// TIA Portal V18 export
VAR_GLOBAL   // PLC tag table "默认变量表"
   Room1_ES1 AT %I200.0 : Bool;
   Room1_ES2 AT %I200.1 : Bool;
   Room1_ES3 AT %I200.2 : Bool;
   Room1_ES4 AT %I200.3 : Bool;
   Room1_ES5 AT %I206.0 : Bool;
   Room1Control_ES6 AT %I206.1 : Bool;
   "Room1_Key1.1" AT %I206.2 : Bool;
   "Room1Control_Key1.1" AT %I206.3 : Bool;
   "Room1_door1.1" AT %I212.0 : Bool;
   Room2_ES1 AT %I218.0 : Bool;
   Room2_ES2 AT %I218.1 : Bool;
   Room2_ES3 AT %I218.2 : Bool;
   Room2_ES4 AT %I218.3 : Bool;
   Room2_ES5 AT %I224.0 : Bool;
   Room2Control_ES6 AT %I224.1 : Bool;
   "Room2_Key1.1" AT %I224.2 : Bool;
   "Room2Control_Key1.1" AT %I224.3 : Bool;
   "Room2_door1.1" AT %I230.0 : Bool;
   ACC_ES1 AT %I236.0 : Bool;
   ACC_ES2 AT %I236.1 : Bool;
   ACC_ES3 AT %I236.2 : Bool;
   ACC_ES4 AT %I236.3 : Bool;
   "ACC_Key1.1" AT %I242.2 : Bool;
   "ACCControl_Key1.1" AT %I242.3 : Bool;
   "ACC_door1.1" AT %I248.0 : Bool;
   "ACC_door2.1" AT %I248.1 : Bool;
   VerticalBeam_ES1 AT %I254.0 : Bool;   // vertical beam ES
   VerticalBeam_ES2 AT %I254.1 : Bool;
   VerticalBeam_ES3 AT %I254.2 : Bool;
   VerticalBeam_ES4 AT %I254.3 : Bool;
   "VerticalBeam_Key1.1" AT %I260.2 : Bool;
   "VerticalBeamControl_Key1.1" AT %I260.3 : Bool;
   "VerticalBeam_door1.1" AT %I266.0 : Bool;
   "VerticalBeam_door2.1" AT %I266.1 : Bool;
   Room1_SB1 AT %I100.0 : Bool;   // 搜索清场按钮1
   Room1_SB2 AT %I100.1 : Bool;
   Room2_SB1 AT %I100.4 : Bool;
   Room2_SB2 AT %I100.5 : Bool;
   ACC_SB1 AT %I101.0 : Bool;
   ACC_SB2 AT %I101.1 : Bool;
   VerticalBeam_SB1 AT %I101.4 : Bool;
   VerticalBeam_SB2 AT %I101.5 : Bool;
   ACC_Ready AT %I102.0 : Bool;
   ACC_Run AT %I102.1 : Bool;
   ACC_StopBeam AT %I102.2 : Bool;
   ACC_Stop AT %I102.3 : Bool;
   ACC_Fault AT %I102.4 : Bool;
   ACC_Mode1 AT %I102.5 : Bool;   // 治疗室1、加速器2、垂直束
   ACC_Mode2 AT %I102.6 : Bool;   // 治疗室2、加速器2、垂直束
   ACC_Mode3 AT %I102.7 : Bool;   // 加速器2、垂直束
   EnvironmentalMonitoring1 AT %I103.4 : Bool;
   EnvironmentalMonitoring2 AT %I103.5 : Bool;
   EnvironmentalMonitoring3 AT %I103.6 : Bool;
   EnvironmentalMonitoring4 AT %I103.7 : Bool;
   Room1_AudibleAlarm AT %Q100.0 : Bool;
   Room1_StrobeLamp1 AT %Q100.1 : Bool;
   Room1_StrobeLamp2 AT %Q100.2 : Bool;
   Room1_Red AT %Q100.5 : Bool;   // 禁止进入指示灯
   Room1_Yellow AT %Q100.6 : Bool;   // 限制进入指示灯
   Room1_Green AT %Q100.7 : Bool;   // 控制进入指示灯
   Room1_Door1NoEntry AT %Q101.0 : Bool;   // 门禁1禁止进入
   Room1_Door1RestrictedEntry AT %Q101.1 : Bool;   // 门禁1限制进入
   Room1_Door1ControlEntry AT %Q101.2 : Bool;   // 门禁1控制进入
   "Room1_door1.2" AT %I212.4 : Bool;
   "Room1_Key1.2" AT %I206.6 : Bool;
   "Room1Control_Key1.2" AT %I206.7 : Bool;
   "Room2_Key1.2" AT %I224.6 : Bool;
   "Room2Control_Key1.2" AT %I224.7 : Bool;
   "Room2_door1.2" AT %I230.4 : Bool;
   "ACC_Key1.2" AT %I242.6 : Bool;
   "ACCControl_Key1.2" AT %I242.7 : Bool;
   "VerticalBeam_Key1.2" AT %I260.6 : Bool;
   "VerticalBeamControl_Key1.2" AT %I260.7 : Bool;
   "VerticalBeam_door1.2" AT %I266.4 : Bool;
   "VerticalBeam_door2.2" AT %I266.5 : Bool;
   "ACC_door1.2" AT %I248.4 : Bool;
   "ACC_door2.2" AT %I248.5 : Bool;
   ACC_Interlock1 AT %Q400.0 : Bool;
   ACC_Interlock2 AT %Q400.1 : Bool;
   RF_Interlock1 AT %Q400.2 : Bool;
   RF_Interlock2 AT %Q400.3 : Bool;
   IonSource_Interlock1 AT %Q400.4 : Bool;
   IonSource_Interlock2 AT %Q400.5 : Bool;
   MIS__Interlock1 AT %Q400.6 : Bool;
   MIS__Interlock2 AT %Q400.7 : Bool;
   Room1_ES1_ValueStatus AT %I201.0 : Bool;
   Room1_ES2_ValueStatus AT %I201.1 : Bool;
   Room1_ES3_ValueStatus AT %I201.2 : Bool;
   Room1_ES4_ValueStatus AT %I201.3 : Bool;
   Room1_ES5_ValueStatus AT %I207.0 : Bool;
   Room1Control_ES6_ValueStatus AT %I207.1 : Bool;
   "Room1_Key1.1_ValueStatus" AT %I207.2 : Bool;
   "Room1Control_Key1.1_ValueStatus" AT %I207.3 : Bool;
   "Room1_Key1.2_ValueStatus" AT %I207.6 : Bool;
   "Room1Control_Key1.2_ValueStatus" AT %I207.7 : Bool;
   "Room1_door1.1_ValueStatus" AT %I213.0 : Bool;
   "Room1_door1.2_ValueStatus" AT %I213.4 : Bool;
   Room2_ES1_ValueStatus AT %I219.0 : Bool;
   Room2_ES2_ValueStatus AT %I219.1 : Bool;
   Room2_ES3_ValueStatus AT %I219.2 : Bool;
   Room2_ES4_ValueStatus AT %I219.3 : Bool;
   Room2_ES5_ValueStatus AT %I225.0 : Bool;
   Room2Control_ES6_ValueStatus AT %I225.1 : Bool;
   "Room2_Key1.1_ValueStatus" AT %I225.2 : Bool;
   "Room2Control_Key1.1_ValueStatus" AT %I225.3 : Bool;
   "Room2_Key1.2_ValueStatus" AT %I225.6 : Bool;
   "Room2Control_Key1.2_ValueStatus" AT %I225.7 : Bool;
   "Room2_door1.1_ValueStatus" AT %I231.0 : Bool;
   "Room2_door1.2_ValueStatus" AT %I231.4 : Bool;
   ACC_ES1_ValueStatus AT %I237.0 : Bool;
   ACC_ES2_ValueStatus AT %I237.1 : Bool;
   ACC_ES3_ValueStatus AT %I237.2 : Bool;
   ACC_ES4_ValueStatus AT %I237.3 : Bool;
   "ACC_Key1.1_ValueStatus" AT %I243.2 : Bool;
   "ACCControl_Key1.1_ValueStatus" AT %I243.3 : Bool;
   "ACC_Key1.2_ValueStatus" AT %I243.6 : Bool;
   "ACCControl_Key1.2_ValueStatus" AT %I243.7 : Bool;
   "ACC_door1.1_ValueStatus" AT %I249.0 : Bool;
   "ACC_door2.1_ValueStatus" AT %I249.1 : Bool;
   "ACC_door1.2_ValueStatus" AT %I249.4 : Bool;
   "ACC_door2.2_ValueStatus" AT %I249.5 : Bool;
   VerticalBeam_ES1_ValueStatus AT %I255.0 : Bool;
   VerticalBeam_ES2_ValueStatus AT %I255.1 : Bool;
   VerticalBeam_ES3_ValueStatus AT %I255.2 : Bool;
   VerticalBeam_ES4_ValueStatus AT %I255.3 : Bool;
   "VerticalBeam_Key1.1_ValueStatus" AT %I261.2 : Bool;
   "VerticalBeamControl_Key1.1_ValueStatus" AT %I261.3 : Bool;
   "VerticalBeam_Key1.2_ValueStatus" AT %I261.6 : Bool;
   "VerticalBeamControl_Key1.2_ValueStatus" AT %I261.7 : Bool;
   "VerticalBeam_door1.1_ValueStatus" AT %I267.0 : Bool;
   "VerticalBeam_door2.1_ValueStatus" AT %I267.1 : Bool;
   "VerticalBeam_door1.2_ValueStatus" AT %I267.4 : Bool;
   "VerticalBeam_door2.2_ValueStatus" AT %I267.5 : Bool;
   ACC_Interlock1_ValueStatus AT %I400.0 : Bool;
   ACC_Interlock2_ValueStatus AT %I400.1 : Bool;
   RF_Interlock1_ValueStatus AT %I400.2 : Bool;
   RF_Interlock2_ValueStatus AT %I400.3 : Bool;
   IonSource_Interlock1_ValueStatus AT %I400.4 : Bool;
   IonSource_Interlock2_ValueStatus AT %I400.5 : Bool;
   MIS__Interlock1_ValueStatus AT %I400.6 : Bool;
   MIS__Interlock2_ValueStatus AT %I400.7 : Bool;
   Room2_AudibleAlarm AT %Q102.0 : Bool;
   Room2_StrobeLamp1 AT %Q102.1 : Bool;
   Room2_StrobeLamp2 AT %Q102.2 : Bool;
   Room2_Red AT %Q102.5 : Bool;
   Room2_Yellow AT %Q102.6 : Bool;
   Room2_Green AT %Q102.7 : Bool;
   Room2_Door1NoEntry AT %Q103.0 : Bool;
   Room2_Door1RestrictedEntry AT %Q103.1 : Bool;
   Room2_Door1ControlEntry AT %Q103.2 : Bool;
   ACC_AudibleAlarm AT %Q104.0 : Bool;
   ACC_StrobeLamp1 AT %Q104.1 : Bool;
   ACC_StrobeLamp2 AT %Q104.2 : Bool;
   ACC_Red AT %Q104.5 : Bool;
   ACC_Yellow AT %Q104.6 : Bool;
   ACC_Green AT %Q104.7 : Bool;
   ACC_StrobeLamp3 AT %Q104.3 : Bool;
   ACC_StrobeLamp4 AT %Q104.4 : Bool;
   ACC_Door1NoEntry AT %Q105.0 : Bool;
   ACC_Door1RestrictedEntry AT %Q105.1 : Bool;
   ACC_Door1ControlEntry AT %Q105.2 : Bool;
   ACC_Door2NoEntry AT %Q105.3 : Bool;
   ACC_Door2RestrictedEntry AT %Q105.4 : Bool;
   ACC_Door2ControlEntry AT %Q105.5 : Bool;
   VerticalBeam_AudibleAlarm AT %Q106.0 : Bool;
   VerticalBeam_StrobeLamp1 AT %Q106.1 : Bool;
   VerticalBeam_StrobeLamp2 AT %Q106.2 : Bool;
   VerticalBeam_StrobeLamp3 AT %Q106.3 : Bool;
   VerticalBeam_StrobeLamp4 AT %Q106.4 : Bool;
   VerticalBeam_Red AT %Q106.5 : Bool;
   VerticalBeam_Yellow AT %Q106.6 : Bool;
   VerticalBeam_Green AT %Q106.7 : Bool;
   VerticalBeam_Door1NoEntry AT %Q107.0 : Bool;
   VerticalBeam_Door1RestrictedEntry AT %Q107.1 : Bool;
   VerticalBeam_Door1ControlEntry AT %Q107.2 : Bool;
   VerticalBeam_Door2NoEntry AT %Q107.3 : Bool;
   VerticalBeam_Door2RestrictedEntry AT %Q107.4 : Bool;
   VerticalBeam_Door2ControlEntry AT %Q107.5 : Bool;
   Room1_AreaReady AT %Q108.0 : Bool;   // 治疗室1控制区就绪
   Room2_AreaReady AT %Q108.1 : Bool;   // 治疗室2控制区就绪
   ACC_AreaReady AT %Q108.2 : Bool;   // 加速器2控制区就绪
   Room1_StartAlarm AT %Q101.7 : Bool;
   Room2_StartAlarm AT %Q103.7 : Bool;
   ACC_StartAlarm AT %Q105.7 : Bool;
   VerticalBeam_StartAlarm AT %Q107.7 : Bool;
   Room1_BeamAllowed AT %Q108.4 : Bool;   // 允许治疗室1打靶
   Room2_BeamAllowed AT %Q108.5 : Bool;   // 允许治疗室2打靶
   ACC_BeamAllowed AT %Q108.6 : Bool;   // 允许加速器出束
   VerticalBeam_AreaReady AT %Q108.3 : Bool;   // 垂直束控制区就绪
END_VAR
